TYPE ST_RejectReasonOUT2 :
STRUCT
	Reason	:STRING;
END_STRUCT
END_TYPE

(* stored: Version 1.1.0.1, ProductVersion 3.1.4024.13
   DUT ST_RejectReasonOUT2: Id {5ba5908c-3fe6-4306-8980-620de402a868} *)
